(* PLC project KinIn_v3.project, CODESYS CODESYS V3.5 SP19 *)
(* stored: creationDateTime 2025-01-20T16:22:39.8484232, modificationDateTime 2025-01-20T16:17:39.6822999 *)

FUNCTION_BLOCK pInv
  VAR_INPUT
    matrix : ARRAY[1..GVL.pInv_dim1, 1..GVL.pInv_dim2] OF REAL;
  END_VAR
  VAR_OUTPUT
    pInvMatrix : ARRAY[1..GVL.pInv_dim2, 1..GVL.pInv_dim1] OF REAL;
  END_VAR
  VAR
    transpose : transpose;
    MatMul : MatMul;
    Inv : Inv;
    matrixTrans : ARRAY[1..GVL.pInv_dim2, 1..GVL.pInv_dim1] OF REAL;  (* transpose matrix *)
    matSquareSize2 : ARRAY[1..GVL.nInvSize, 1..GVL.nInvSize] OF REAL;  (* matrix with the second size of the original matrix *)
    InverseMatrix : ARRAY[1..GVL.nInvSize, 1..GVL.nInvSize] OF REAL;
  END_VAR

            transpose(B:=matrix , Bt:=matrixTrans );

MatMul(mat1:= matrixTrans, mat2:= matrix, 
	MatResult:= matSquareSize2);

Inv(matSquare:= matSquareSize2, 
	InverseMatrix=> InverseMatrix);
	
MatMul(mat1:= InverseMatrix, mat2:= matrixTrans, 
	MatResult:= pInvMatrix);

          
END_FUNCTION_BLOCK
